TYPE "HU_Tank_Par"
VERSION : 0.1
// Block: HU_Tank_Par
   STRUCT
      DelayCheckFilterClogged : Time;
      DelayRecirculationPumpOff : Time;
      HeatingEnable : Bool;
      HeatingTempRunPermit : Real;
      HeatingSetpoint : Real;
      HeatingUnit2Delta : Real;
      CoolingEnable : Bool;
      CoolingSetpoint : Real;
      WeeklyClockEnable : Bool;
      WeeklyClockSetup : Array[1..7] of WkClockSet;
   END_STRUCT;

END_TYPE
